VAR_GLOBAL CONSTANT
	nEndOfNodeIDVarsArray_3Dim: UINT := 9 ;
	nArrayTestLength_3DimX: UDINT := 4;
	nArrayTestLength_3DimY: UDINT := 2;
	nArrayTestLength_3DimZ: UDINT := 2;
	//nArrayTestLength_3DimX*nArrayTestLength_3DimY*nArrayTestLength_3DimZ*80
	nMaxReadDataArray_3Dim: UDINT := 1280; 
	//sOpcUA_URL: STRING := 'opc.tcp://henningm-nb:4840';
	sOpcUA_URL: STRING := 'opc.tcp://localhost:4842';
	sNodeIDNamespace: STRING := 'TmcPLC';
END_VAR
VAR_GLOBAL
	NodeID_Identifiers: ARRAY[0..nEndOfNodeIDVarsArray_3Dim] OF STRING := 
		['GVL_ArrayTests3DimPLC.stat_BOOL_3Dim', 
		 'GVL_ArrayTests3DimPLC.stat_BSTRARRAY_3Dim',
		 'GVL_ArrayTests3DimPLC.stat_I1_3Dim', 
		 'GVL_ArrayTests3DimPLC.stat_I2_3Dim', 
		 'GVL_ArrayTests3DimPLC.stat_I4_3Dim', 
		 'GVL_ArrayTests3DimPLC.stat_R8_3Dim', 
		 'GVL_ArrayTests3DimPLC.stat_UI1_3Dim', 
		 'GVL_ArrayTests3DimPLC.stat_UI2_3Dim',  
		 'GVL_ArrayTests3DimPLC.stat_UI4_3Dim', 
		 'GVL_ArrayTests3DimPLC.stat_DATE_3Dim'
	];
	NodeID_Sizes: ARRAY[0..nEndOfNodeIDVarsArray_3Dim] OF UDINT := 
		[(1 * nArrayTestLength_3DimX * nArrayTestLength_3DimY * nArrayTestLength_3DimZ), 
		 (81 * nArrayTestLength_3DimX * nArrayTestLength_3DimY * nArrayTestLength_3DimZ), 
		 (1 * nArrayTestLength_3DimX * nArrayTestLength_3DimY * nArrayTestLength_3DimZ), 
		 (2 * nArrayTestLength_3DimX * nArrayTestLength_3DimY * nArrayTestLength_3DimZ), 
		 (4 * nArrayTestLength_3DimX * nArrayTestLength_3DimY  * nArrayTestLength_3DimZ), 
		 (8 * nArrayTestLength_3DimX * nArrayTestLength_3DimY  * nArrayTestLength_3DimZ), 
		 (1 * nArrayTestLength_3DimX * nArrayTestLength_3DimY  * nArrayTestLength_3DimZ), 
		 (2 * nArrayTestLength_3DimX * nArrayTestLength_3DimY  * nArrayTestLength_3DimZ), 
	     (4 * nArrayTestLength_3DimX * nArrayTestLength_3DimY  * nArrayTestLength_3DimZ), 
	     (4 * nArrayTestLength_3DimX * nArrayTestLength_3DimY  * nArrayTestLength_3DimZ)
	];
	NodeID_DoOrDont: ARRAY[0..nEndOfNodeIDVarsArray_3Dim] OF BOOL := 
		[TRUE, //'GVL_ArrayTests3DimPLC.stat_BOOL_3Dim', 
		 TRUE, //'GVL_ArrayTests3DimPLC.stat_BSTRARRAY_3Dim',
		 TRUE, //'GVL_ArrayTests3DimPLC.stat_I1_3Dim', 
		 TRUE, //'GVL_ArrayTests3DimPLC.stat_I2_3Dim', 
		 TRUE, //'GVL_ArrayTests3DimPLC.stat_I4_3Dim', 
		 TRUE, //'GVL_ArrayTests3DimPLC.stat_R8_3Dim', 
		 TRUE, //'GVL_ArrayTests3DimPLC.stat_UI1_3Dim', 
		 TRUE, //'GVL_ArrayTests3DimPLC.stat_UI2_3Dim',  
		 TRUE, //'GVL_ArrayTests3DimPLC.stat_UI4_3Dim', 
		 FALSE //'GVL_ArrayTests3DimPLC.stat_DATE_3Dim'
	];
	NodeID_WriteCommands: ARRAY[0..nEndOfNodeIDVarsArray_3Dim] OF U_Arrays3DimInOne := [
			(bBool := [TRUE, FALSE, TRUE, FALSE, TRUE, FALSE, TRUE, FALSE, TRUE, FALSE, TRUE, FALSE, TRUE, FALSE, TRUE, FALSE]), 
	 		(sString := ['aaa', 'bbbb', 'ccccc', 'ddddddd', 'aaa', 'bbbb', 'ccccc', 'ddddddd', 'aaa', 'bbbb', 'ccccc', 'ddddddd', 'aaa', 'bbbb', 'ccccc', 'ddddddd']), 
			(bByte := [123, 124, 125, 126, 123, 124, 125, 126, 123, 124, 125, 126, 123, 124, 125, 126]), 
			(nInt := [127, 128, 129, 130,127, 128, 129, 130, 127, 128, 129, 130,127, 128, 129, 130]), 
			(nUdint := [131, 132, 133, 134, 131, 132, 133, 134, 131, 132, 133, 134, 131, 132, 133, 134]), 
			(nLReal := [1.23456, 1.23457, 1.23458, 1.23459, 1.23456, 1.23457, 1.23458, 1.23459, 1.23456, 1.23457, 1.23458, 1.23459, 1.23456, 1.23457, 1.23458, 1.23459]), 
			(bByte := [111, 112, 113, 114, 111, 112, 113, 114, 111, 112, 113, 114, 111, 112, 113, 114]), 
			(nInt := [115, 116, 117, 118,115, 116, 117, 118, 115, 116, 117, 118,115, 116, 117, 118]), 
			(nUdint := [119, 120, 121, 122, 119, 120, 121, 122, 119, 120, 121, 122, 119, 120, 121, 122]), 
			(dDate := [DT#2008-9-26-0:11:12, DT#2008-9-26-0:11:13, DT#2008-9-26-0:11:14, DT#2008-9-26-0:11:15, DT#2008-9-26-0:11:12, DT#2008-9-26-0:11:13, DT#2008-9-26-0:11:14, DT#2008-9-26-0:11:15, DT#2008-9-26-0:11:12, DT#2008-9-26-0:11:13, DT#2008-9-26-0:11:14, DT#2008-9-26-0:11:15, DT#2008-9-26-0:11:12, DT#2008-9-26-0:11:13, DT#2008-9-26-0:11:14, DT#2008-9-26-0:11:15]) 
	];
	NodeID_ReadResults: ARRAY[0..nEndOfNodeIDVarsArray_3Dim] OF U_Arrays3DimInOne;
	NodeID_ReadWrittenResults: ARRAY[0..nEndOfNodeIDVarsArray_3Dim] OF U_Arrays3DimInOne;
	NodeID_CheckReadWrite: ARRAY[0..nEndOfNodeIDVarsArray_3Dim] OF BOOL;
	
	//Data fields
	test : BOOL; (*~ (OPC : 1 : enabled for OPC) *)
	stat_BOOL_3Dim: 		ARRAY[1..nArrayTestLength_3DimX, 1..nArrayTestLength_3DimY, 1..nArrayTestLength_3DimZ] OF BOOL 	:= [TRUE, TRUE, TRUE, TRUE, FALSE, FALSE, FALSE, FALSE,TRUE, TRUE, TRUE, TRUE, FALSE, FALSE, FALSE, FALSE]; 						(*~ (OPC : 1 : enabled for OPC) *)
	stat_BSTRARRAY_3Dim: 	ARRAY[1..nArrayTestLength_3DimX, 1..nArrayTestLength_3DimY, 1..nArrayTestLength_3DimZ] OF STRING 	:= ['these', 'are', 'init', 'values', 'which', 'will', 'be', 'overwritten', 'these', 'are', 'init', 'values', 'which', 'will', 'be', 'overwritten'];	(*~ (OPC : 1 : enabled for OPC) *)
	stat_I1_3Dim: 			ARRAY[1..nArrayTestLength_3DimX, 1..nArrayTestLength_3DimY, 1..nArrayTestLength_3DimZ] OF BYTE		:= [1, 1, 1, 1, 1, 1, 1, 1, 1, 1, 1, 1, 1, 1, 1, 1];													(*~ (OPC : 1 : enabled for OPC) *)
	stat_I2_3Dim: 			ARRAY[1..nArrayTestLength_3DimX, 1..nArrayTestLength_3DimY, 1..nArrayTestLength_3DimZ] OF INT		:= [1, 1, 1, 1, 1, 1, 1, 1, 1, 1, 1, 1, 1, 1, 1, 1];													(*~ (OPC : 1 : enabled for OPC) *)
	stat_I4_3Dim:			ARRAY[1..nArrayTestLength_3DimX, 1..nArrayTestLength_3DimY, 1..nArrayTestLength_3DimZ] OF DINT 	:= [1, 1, 1, 1, 1, 1, 1, 1, 1, 1, 1, 1, 1, 1, 1, 1];													(*~ (OPC : 1 : enabled for OPC) *)
	stat_R8_3Dim: 			ARRAY[1..nArrayTestLength_3DimX, 1..nArrayTestLength_3DimY, 1..nArrayTestLength_3DimZ] OF LREAL	:= [1.1, 1.1, 1.1, 1.1, 1.1, 1.1, 1.1, 1.1, 1.1, 1.1, 1.1, 1.1, 1.1, 1.1, 1.1, 1.1];									(*~ (OPC : 1 : enabled for OPC) *)
	stat_UI1_3Dim:			ARRAY[1..nArrayTestLength_3DimX, 1..nArrayTestLength_3DimY, 1..nArrayTestLength_3DimZ] OF BYTE		:= [1, 1, 1, 1, 1, 1, 1, 1, 1, 1, 1, 1, 1, 1, 1, 1];													(*~ (OPC : 1 : enabled for OPC) *)
	stat_UI2_3Dim: 			ARRAY[1..nArrayTestLength_3DimX, 1..nArrayTestLength_3DimY, 1..nArrayTestLength_3DimZ] OF UINT		:= [1, 1, 1, 1, 1, 1, 1, 1, 1, 1, 1, 1, 1, 1, 1, 1];													(*~ (OPC : 1 : enabled for OPC) *)
	stat_UI4_3Dim: 			ARRAY[1..nArrayTestLength_3DimX, 1..nArrayTestLength_3DimY, 1..nArrayTestLength_3DimZ] OF UDINT	:= [1, 1, 1, 1, 1, 1, 1, 1,1, 1, 1, 1, 1, 1, 1, 1];													(*~ (OPC : 1 : enabled for OPC) *)
	stat_DATE_3Dim:			ARRAY[1..nArrayTestLength_3DimX, 1..nArrayTestLength_3DimY, 1..nArrayTestLength_3DimZ] OF DT	:= [DT#2014-2-20-0:11:12, DT#2014-2-20-0:11:12, DT#2014-2-20-0:11:12, DT#2014-2-20-0:11:12, DT#2014-2-20-0:11:12, DT#2014-2-20-0:11:12, DT#2014-2-20-0:11:12, DT#2014-2-20-0:11:12, DT#2014-2-20-0:11:12, DT#2014-2-20-0:11:12, DT#2014-2-20-0:11:12, DT#2014-2-20-0:11:12, DT#2014-2-20-0:11:12, DT#2014-2-20-0:11:12, DT#2014-2-20-0:11:12, DT#2014-2-20-0:11:12];													(*~ (OPC : 1 : enabled for OPC) *)
		
END_VAR

(* stored: Version 1.1.0.1, ProductVersion 3.1.0.24
   GVL GVL_ArrayTests3DimPLC: Id {9856cb8e-f08c-48bb-8834-2e42519f0200} *)
